// TIA Portal V16 export
// export: Created 2020-02-19T17:17:18.4449535Z, ExportSetting WithDefaults, WithReadOnly, DisplayName Totally Integrated Automation Portal, DisplayVersion V16, DisplayName TIA Portal Version Control Interface, DisplayVersion V16, DisplayName TIA Portal Openness, DisplayVersion V16, DisplayName STEP 7 Professional, DisplayVersion V16, DisplayName STEP 7 Safety, DisplayVersion V16, DisplayName WinCC Advanced, DisplayVersion V16
FUNCTION "TestFC1" : Void   // FC3, LAD
{ S7_Optimized_Access := 'TRUE' }
VERSION : 0.1
// stored: AutoNumber true, CodeModifiedDate 2020-02-19T17:12:50.997434Z, CompileDate 2020-02-19T17:16:33.8926525Z, CreationDate 2020-02-19T17:12:22.7008022Z, HandleErrorsWithinBlock false, InterfaceModifiedDate 2020-02-19T17:12:22.7008022Z, IsConsistent true, IsIECCheckEnabled false, IsKnowHowProtected false, IsWriteProtected false, LibraryConformanceStatus Das Objekt ist bibliothekskonform., ModifiedDate 2020-02-19T17:12:56.1537805Z, ParameterModified 2020-02-19T17:12:22.7008022Z, PLCSimAdvancedSupport true, SetENOAutomatically false, StructureModified 2020-02-19T17:12:22.7008022Z, UDAEnableTagReadback false
BEGIN

REGION Network 1: Netz 1
END_REGION

REGION Network 2: Netz 2
END_REGION
END_FUNCTION
